// TIA Portal V20 export
TYPE "LConSMC_typeSyncDynamics"
// [Einheit der Achse] Dynamiken zum synchronisieren auf eine laufende Bahn  Wirksam wenn "enable" & "speedMatch" = TRUE / [Unit of the axis] Dynamics for synchronizing to line speed  Active if "enable" & "speedMatch" = TRUE
// stored: Access Published
   STRUCT
      acceleration : Real := -1.0;   // Beschleunigung in Achseinheit / Acceleration value: Units are taken from the TO
      deceleration : Real := -1.0;   // Verzögerung in Achseinheit / Deceleration value: Units are taken from the TO
      jerk : Real := -1.0;   // Ruckbegrenzung in Achseinheit / Jerk value : Units are taken from the TO
      abortAcceleration : Bool := FALSE;   // TRUE: Setze aktuelle Beschleunigung auf 0 FALSE: Baue aktuelle Beschleunigung über konfigurierten Ruck ab / TRUE: Abort acceleration immediately, FALSE: Reduce current acceleration via Jerk
      syncToleranceFactor : Real := 1.0;   // Faktor zum Anpassen der Synchronisationstoleranz / Factor to adjust synchronization tolerance
   END_STRUCT;
END_TYPE
